// TIA Portal V17 export
// export: Created 2026-10-01T22:10:11.4871335Z, ExportSetting WithDefaults, DisplayName Totally Integrated Automation Portal, DisplayVersion V17, DisplayName TIA Portal Openness, DisplayVersion V17, DisplayName TIA Portal Version Control Interface, DisplayVersion V17, DisplayName SINAMICS Startdrive Advanced, DisplayVersion V17, DisplayName SINAMICS Startdrive G130, G150, S120, S150, SINAMICS MV, G220, S200, S210, DisplayVersion V17, DisplayName SINAMICS Startdrive G110M, G120, G120C, G120D, G120P, G115D, DisplayVersion V17, DisplayName STEP 7 Professional, DisplayVersion V17, DisplayName STEP 7 Safety, DisplayVersion V17, DisplayName WinCC Basic/Comfort/Advanced, DisplayVersion V17, DisplayName WinCC Unified, DisplayVersion V17
FUNCTION_BLOCK "ZZ_LadTest_Scale"   // FB29, LAD
{ S7_Optimized_Access := 'TRUE' }
VERSION : 0.1
// stored: AutoNumber true, IsIECCheckEnabled false, IsRetainMemResEnabled false, MemoryReserve 100, SetENOAutomatically false, UDAEnableTagReadback false
   VAR_INPUT
      Start : Bool;
      "A" : Int;
      "B" : Int;
      X : Real;
   END_VAR
   VAR
      R1 : Int;
      R2 : Int;
      R3 : Int;
      R4 : Int;
      R5 : Int;
      Nrm : Real;
      Scl : Real;
      Latch : Bool;
      Latch2 : Bool;
   END_VAR
BEGIN

REGION Network 1
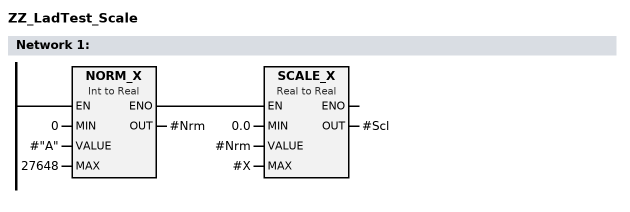
   RUNG wire#powerrail
      { S7_Templates := "[SrcType := Int, DestType := Real]" } Normalize(min := 0, value := #"A", max := 27648, out => #Nrm)
      { S7_Templates := "[SrcType := Real, DestType := Real]" } Scale(min := 0.0, value := #Nrm, max := #X, out => #Scl)
   END_RUNG
   // the same network as SCL:
   #Nrm := NORM_X(MIN := 0, VALUE := #"A", MAX := 27648);
   #Scl := SCALE_X(MIN := 0.0, VALUE := #Nrm, MAX := #X);
END_REGION
END_FUNCTION_BLOCK
